// TIA Portal project "DairyPLant" (V14)
// A SCADA system for monitoring a small scale Dairy Plant

(* hardware
DEVICE "Plant Station"  SIMATIC PC station
   slot 0: "SIMATIC PC station"  Rail  SIMATIC PC-Station  V1.0
      slot 125: "Stationmanager"  Station_Manager  V6.0.4
   slot 1: "PLant"  WinCC RT Professional  6AV2 105-0xxxx-xxxx  14.0.1.0
*)

(* ===== HMI "PLant" =====
system functions are stored by id; their names below are inferred from use

HMI tags "Default tag table"
   "IndusysLTD" : String[10], internal   // Indusys LTD website

HMI tags "Boiler"
   "Boiler_ON/OFF" : Bool, internal

screen "Storage Tanks (Raw Milk)" 1920x1080
   GraphicView "Graphic view_1" at 8,7 size 120x118; Picture "Indusys"
      on Click: ActivateScreen("Home", 0)
   Group "Group" at 230,249 size 374x718; Picture "Graphic_20"
   GraphicView "Graphic view_3" at 230,574 size 127x84; Picture "Graphic_20"
   GraphicView "Graphic view_2" at 316,249 size 288x718; Picture "Graphic_19"

screen "Storage Tanks (Water-Raw)" 1920x1080
   GraphicView "Graphic view_1" at 8,7 size 120x118; Picture "Indusys"
      on Click: ActivateScreen("Home", 0)
   Group "Group_1" at 630,93 size 145x208; Picture "Graphic_4"
   GraphicView "Graphic view_4" at 639,93 size 125x204; Picture "Graphic_4"
   Bar "Bar_1" at 630,117 size 145x184; MinimumValue 0; MaximumValue 100

screen "Storage Tanks (Pasteurized Milk)" 1920x1080
   GraphicView "Graphic view_1" at 8,7 size 120x118; Picture "Indusys"
      on Click: ActivateScreen("Home", 0)
   Group "Group" at 230,249 size 374x718; Picture "Graphic_20"
   GraphicView "Graphic view_3" at 230,574 size 127x84; Picture "Graphic_20"
   GraphicView "Graphic view_2" at 316,249 size 288x718; Picture "Graphic_19"

screen "Storage (Culture Room)" 1920x1080
   GraphicView "Graphic view_1" at 8,7 size 120x118; Picture "Indusys"
      on Click: ActivateScreen("Home", 0)
   GraphicView "Graphic view_2" at 110,175 size 168x167; Picture "Graphic_18"

screen "Storage (Cold Room)" 1920x1080
   GraphicView "Graphic view_1" at 8,7 size 120x118; Picture "Indusys"
      on Click: ActivateScreen("Home", 0)

screen "Sterilizer" 1920x1080
   GraphicView "Graphic view_1" at 8,7 size 120x118; Picture "Indusys"
      on Click: ActivateScreen("Home", 0)
   GraphicView "Graphic view_2" at 96,170 size 137x141; Picture "Graphic_18"

screen "CIP" 1920x1080
   GraphicView "Graphic view_1" at 8,7 size 120x118; Picture "Indusys"
      on Click: ActivateScreen("Home", 0)
   Group "Group" at 176,150 size 188x345; Picture "Graphic_8"
   GraphicView "Graphic view_2" at 184,150 size 169x345; Picture "Graphic_8"
   Bar "Bar_1" at 176,170 size 188x139

screen "KPLC" 1920x1080
   GraphicView "Graphic view_1" at 8,7 size 120x118; Picture "Indusys"
      on Click: ActivateScreen("Home", 0)
   GraphicView "Graphic view_2" at 88,145 size 259x211; Picture "Graphic_16"
   GraphicView "Graphic view_3" at 382,245 size 119x122; Picture "Graphic_17"

screen "Homogenizer (Stage 2)" 1920x1080
   GraphicView "Graphic view_1" at 8,7 size 120x118; Picture "Indusys"
      on Click: ActivateScreen("Home", 0)
   GraphicView "Graphic view_2" at 230,209 size 325x317; Picture "Graphic_14"

screen "Homogenizer (Stage 1)" 1920x1080
   GraphicView "Graphic view_1" at 8,7 size 120x118; Picture "Indusys"
      on Click: ActivateScreen("Home", 0)
   GraphicView "Graphic view_2" at 366,274 size 231x234; Picture "Graphic_14"

screen "Generator" 1920x1080
   GraphicView "Graphic view_1" at 8,7 size 120x118; Picture "Indusys"
      on Click: ActivateScreen("Home", 0)
   GraphicView "Graphic view_2" at 275,170 size 318x179; Picture "Graphic_13"

screen "Filling Machine" 1920x1080
   GraphicView "Graphic view_1" at 8,7 size 120x118; Picture "Indusys"
      on Click: ActivateScreen("Home", 0)
   GraphicView "Graphic view_2" at 158,101 size 466x307; Picture "Graphic_12"

screen "Diesel Tank" 1920x1080
   GraphicView "Graphic view_1" at 8,7 size 120x118; Picture "Indusys"
      on Click: ActivateScreen("Home", 0)
   GraphicView "Graphic view_2" at 141,148 size 315x193; Picture "Graphic_11"

screen "Cream Seperator" 1920x1080
   GraphicView "Graphic view_1" at 8,7 size 120x118; Picture "Indusys"
      on Click: ActivateScreen("Home", 0)
   GraphicView "Graphic view_2" at 341,277 size 263x224; Picture "Graphic_10"

screen "Cooling Towers" 1920x1080
   GraphicView "Graphic view_1" at 8,7 size 120x118; Picture "Indusys"
      on Click: ActivateScreen("Home", 0)
   GraphicView "Graphic view_2" at 547,125 size 521x602; Picture "Graphic_9"

screen "Chiller" 1920x1080
   GraphicView "Graphic view_1" at 8,7 size 120x118; Picture "Indusys"
      on Click: ActivateScreen("Home", 0)
   GraphicView "Graphic view_2" at 260,238 size 432x466; Picture "Graphic_5"

screen "Boiler" 1920x1080
   GraphicView "Graphic view_1" at 8,7 size 120x118; Picture "Indusys"
      on Click: ActivateScreen("Home", 0)
   Group "Group" at 141,147 size 370x242; Picture "Graphic_2"
   Group "Group_1" at 630,93 size 145x208; Picture "Graphic_4"
   GraphicView "Graphic view_2" at 141,147 size 370x242; Picture "Graphic_2"
   GraphicView "Graphic view_3" at 267,305 size 234x53; Picture "Graphic_3"
      PropertyAnimation0 <- "Boiler_ON/OFF"
   GraphicView "Graphic view_4" at 639,93 size 125x204; Picture "Graphic_4"
   Bar "Bar_1" at 630,117 size 145x184; MinimumValue 0; MaximumValue 100

screen "Air Compressor" 1920x1080
   GraphicView "Graphic view_1" at 8,7 size 120x118; Picture "Indusys"
      on Click: ActivateScreen("Home", 0)
   GraphicView "Graphic view_2" at 157,259 size 178x193; Picture "Graphic_1"
   TextField "Text field_1" at 420,240 size 55x21; Text 'Current'
   TextField "Text field_2" at 420,295 size 55x21; Text 'Voltage'
   TextField "Text field_3" at 420,343 size 61x21; Text 'Capacity'
   TextField "Text field_4" at 420,393 size 56x21; Text 'Volume'
   TextField "Text field_5" at 420,435 size 62x21; Text 'Pressure'
   TextField "Text field_6" at 420,479 size 62x21; Text 'Flowrate'
   TextField "Text field_7" at 420,200 size 38x21; Text 'Make'
   TextField "Text field_8" at 418,521 size 53x21; Text 'Uptime'
   TextField "Text field_9" at 418,585 size 68x21; Text 'Messages'
   TextField "Text field_10" at 412,627 size 46x21; Text 'Power'

screen "UPS" 1920x1080
   GraphicView "Graphic view_1" at 8,7 size 120x118; Picture "Indusys"
      on Click: ActivateScreen("Home", 0)
   GraphicView "Graphic view_2" at 192,382 size 221x299; Picture "Graphic_22"

screen "Home" 1920x1080
   GraphicView "Graphic view_1" at 8,7 size 120x118; Picture "Indusys"
      on Click: ActivateScreen("Home", 0)
   Button "Button_1" at 49,147 size 262x33; TextOff 'Air Compressor'
      on Click: ActivateScreen("Air Compressor", 0)
   Button "Button_2" at 49,200 size 262x33; TextOff 'Boiler'
      on Click: ActivateScreen("Boiler", 0)
   Button "Button_3" at 49,253 size 262x33; TextOff 'Chiller'
      on Click: ActivateScreen("Chiller", 0)
   Button "Button_4" at 49,308 size 262x33; TextOff 'CIP'
      on Click: ActivateScreen("CIP", 0)
   Button "Button_5" at 49,363 size 262x33; TextOff 'Cooling Towers'
      on Click: ActivateScreen("Cooling Towers", 0)
   Button "Button_6" at 49,415 size 262x33; TextOff 'Cream Seperator'
      on Click: ActivateScreen("Cream Seperator", 0)
   Button "Button_7" at 49,474 size 262x33; TextOff 'Diesel Tank'
      on Click: ActivateScreen("Diesel Tank", 0)
   Button "Button_8" at 49,522 size 262x33; TextOff 'Filling Machine'
      on Click: ActivateScreen("Filling Machine", 0)
   Button "Button_9" at 444,147 size 262x33; TextOff 'Generator'
      on Click: ActivateScreen("Generator", 0)
   Button "Button_10" at 444,200 size 262x33; TextOff 'Homogenizer (Stage 1)'
      on Click: ActivateScreen("Homogenizer (Stage 1)", 0)
   Button "Button_11" at 444,255 size 262x33; TextOff 'Homogenizer (Stage 2)'
      on Click: ActivateScreen("Homogenizer (Stage 2)", 0)
   Button "Button_12" at 444,312 size 262x33; TextOff 'KPLC'
      on Click: ActivateScreen("KPLC", 0)
   Button "Button_13" at 444,363 size 262x33; TextOff 'Sterilizer'
      on Click: ActivateScreen("Sterilizer", 0)
   Button "Button_14" at 444,415 size 262x33; TextOff 'Storage (Cold Room)'
      on Click: ActivateScreen("Storage (Cold Room)", 0)
   Button "Button_15" at 444,474 size 262x33; TextOff 'Storage (Culture Room)'
      on Click: ActivateScreen("Storage (Culture Room)", 0)
   Button "Button_16" at 444,522 size 262x33; TextOff 'Storage Tanks (Pasteurized Milk)'
      on Click: ActivateScreen("Storage Tanks (Pasteurized Milk)", 0)
   Button "Button_17" at 839,147 size 262x33; TextOff 'Storage Tanks (Raw Milk)'
      on Click: ActivateScreen("Storage Tanks (Raw Milk)", 0)
   Button "Button_18" at 839,200 size 262x33; TextOff 'Storage Tanks (Water-Raw)'
      on Click: ActivateScreen("Storage Tanks (Water-Raw)", 0)
   Button "Button_19" at 839,255 size 262x33; TextOff 'UPS'
      on Click: ActivateScreen("UPS", 0)
   Button "Button_20" at 839,312 size 262x33; TextOff 'Water Treatment Plant'
      on Click: ActivateScreen("Water Treatment Plant", 0)
   Button "Button_21" at 839,363 size 262x33; TextOff 'Web View'
      on Click: ActivateScreen("Web View", 0)

screen "Web View" 1920x1080
   GraphicView "Graphic view_1" at 8,7 size 120x118; Picture "Indusys"
      on Click: ActivateScreen("Home", 0)
   HTMLBrowser "HTML browser_1" at 8,130 size 1908x945
      Address <- "IndusysLTD"

screen "Water Treatment Plant" 1920x1080
   GraphicView "Graphic view_1" at 8,7 size 120x118; Picture "Indusys"
      on Click: ActivateScreen("Home", 0)
   GraphicView "Graphic view_2" at 234,208 size 461x465; Picture "Graphic_7"

screen "Dashboard" 1920x1080
   Button "Button_1" at 1755,2 size 160x30; TextOff 'Home'
      on Click: ActivateScreen("Home", 0)
   TextField "Text field_1" at 843,314 size 50x21; Text 'Supply'
   TextField "Text field_2" at 843,356 size 68x21; Text 'Weighing'
   TextField "Text field_3" at 845,402 size 85x21; Text 'Dump Tank'
   TextField "Text field_4" at 843,453 size 79x21; Text 'Inline filter'
   TextField "Text field_5" at 845,502 size 43x21; Text 'Pump'
   TextField "Text field_6" at 843,552 size 47x21; Text 'Chiller'
   TextField "Text field_7" at 841,623 size 91x21; Text 'Raw Storage'
   TextField "Text field_8" at 1032,314 size 79x21; Text 'Pasteurizer'
   TextField "Text field_9" at 1032,361 size 121x21; Text 'Cream Seperator'
   TextField "Text field_10" at 1032,414 size 96x21; Text 'Homogenizer'
   TextField "Text field_11" at 1032,481 size 141x21; Text 'Storage Pasteurized'
   TextField "Text field_12" at 943,755 size 63x21; Text 'Sterilizer'
   TextField "Text field_13" at 943,717 size 96x21; Text 'Homogenizer'
   TextField "Text field_14" at 943,812 size 36x21; Text 'Filler'
*)